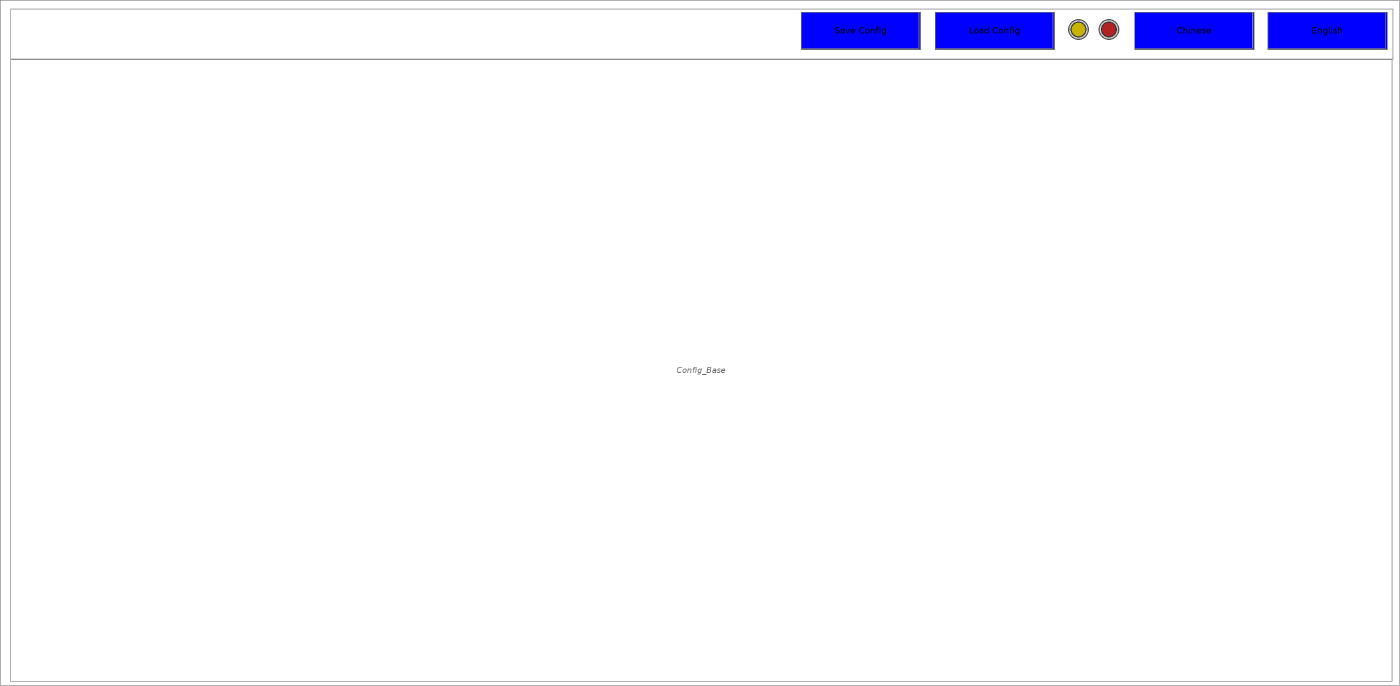
VISUALIZATION Config  // 1755x860
    Frame (13,74 1732x780), input disabled if: gAutoRunningFlag OR gRunningState=RunningStatus.eHomeState
        shows Config_Base()
        shows DataView()
        shows Config_TestSocket()
        shows Config_TXTest()
        shows Config_Coaxial()
        shows Config_RXTest()
        shows Config_UnLoad()
    GroupBox (13,3 1733x71)
        Button (1409,12 150x47), "Chinese"
            OnMouseUp: ChangeLanguage ChangeLanguage=Chinese
            OnMouseUp: execute { gCNErrShow:=TRUE; }
        Button (1576,12 150x47), "English"
            OnMouseUp: ChangeLanguage ChangeLanguage=English
            OnMouseUp: execute { gCNErrShow:=FALSE; }
        Button (1159,12 150x47), "Load Config"
            tap gRead
        Button (991,12 150x47), "Save Config"
            tap gSave
        Lamp1 (1324,19 30x30), variable: DataSave.busy, style: Lamp-Lamp1-Yellow
        Lamp1 (1362,19 30x30), variable: DataSave.error or FB_WStringSave.readError or FB_WStringSave.saveError, style: Lamp-Lamp1-Red
END_VISUALIZATION

(* stored: Version 1.1.0.1, ProductVersion 3.1.4024.12
   Visu Config: Id {c1d77836-4379-4004-a001-32ca207d011c} *)
